{region '#Template'}
	{attribute 'Version' := '1.0.0.0'}
	{attribute 'Tags' := '"LCID": "1031", "Text": "Universal, Control, Scaling"'}
	{attribute 'Tags' := '"LCID": "1033", "Text": "Universal, Control, Scaling"'}
	{attribute 'Description' := '"LCID": "1031", "Text": "Skalierung"'}
	{attribute 'Description' := '"LCID": "1033", "Text": "Scaling"'}
{endregion}
FUNCTION_BLOCK FB_BA_Scale_02 EXTENDS FB_BA_View
VAR_INPUT
	fX			: REAL;
END_VAR
VAR_OUTPUT
	fY			: REAL;
END_VAR
VAR_INPUT CONSTANT
	X1			: FB_BA_AV_Op;	
	X2			: FB_BA_AV_Op;	
	Y1			: FB_BA_AV_Op;	
	Y2			: FB_BA_AV_Op;	
	YMin		: FB_BA_AV_Op;			
	YMax		: FB_BA_AV_Op;											   
	Y			: FB_BA_AV_Op;		
END_VAR
VAR
	Scale		: FB_BA_Chrct02;
END_VAR

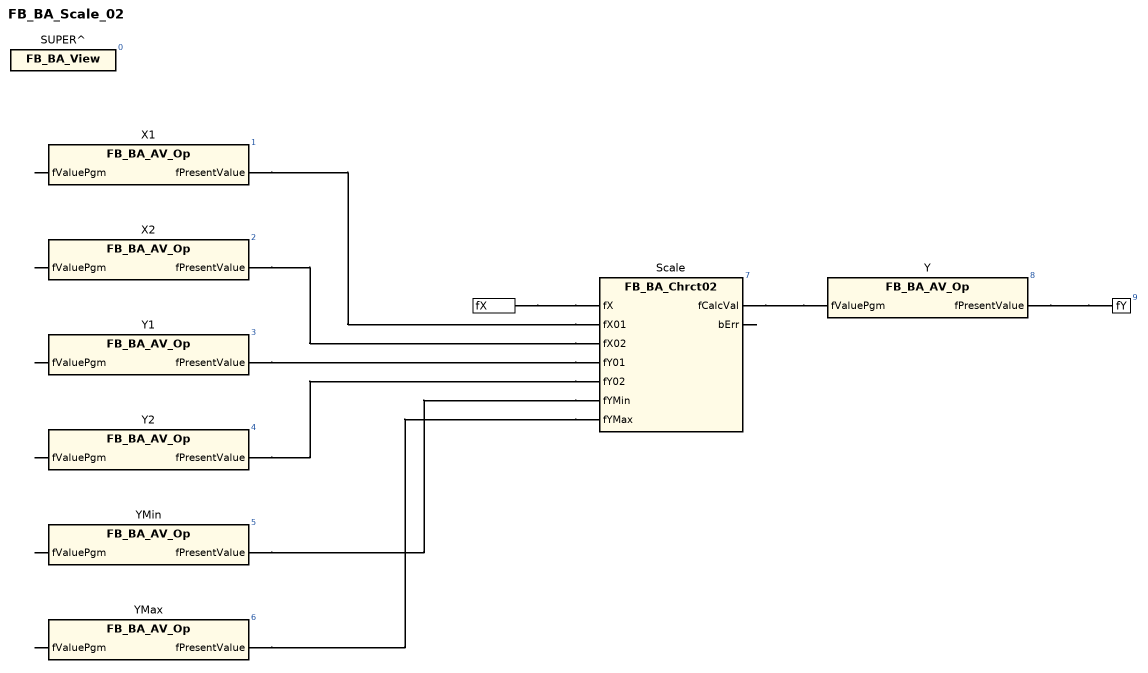
SUPER^(); // FB_BA_View
X1(); // FB_BA_AV_Op
X2(); // FB_BA_AV_Op
Y1(); // FB_BA_AV_Op
Y2(); // FB_BA_AV_Op
YMin(); // FB_BA_AV_Op
YMax(); // FB_BA_AV_Op
Scale(
    fX := fX,
    fX01 := X1.fPresentValue,
    fX02 := X2.fPresentValue,
    fY01 := Y1.fPresentValue,
    fY02 := Y2.fPresentValue,
    fYMin := YMin.fPresentValue,
    fYMax := YMax.fPresentValue); // FB_BA_Chrct02
Y(fValuePgm := Scale.fCalcVal); // FB_BA_AV_Op
fY := Y.fPresentValue;

METHOD FB_init : BOOL
VAR_INPUT
	bInitRetains : BOOL; // if TRUE, the retain variables are initialized (warm start / cold start)
	bInCopyCode : BOOL;  // if TRUE, the instance afterwards gets moved into the copy code (online change)
END_VAR
X1.iParent			:= THIS^;
X1.iLabel			:= LblUniControl.Scale_X01;	
X1.sObjectName		:= '{Idx=01}';		
X1.eUnit			:= E_BA_Unit.eTemperature_DegreesCelsius;						 	 
X1.fValueRm			:= -10.0;
X1.fCOVIncrement	:= BA2_Param.fDefCOVIncrement;		

X2.iParent			:= THIS^;
X2.iLabel			:= LblUniControl.Scale_X02;							
X2.sObjectName		:= '{Idx=02}';								 	 
X2.eUnit			:= E_BA_Unit.eTemperature_DegreesCelsius;						 	 
X2.fValueRm			:= -20.0;
X2.fCOVIncrement	:= BA2_Param.fDefCOVIncrement;		

Y1.iParent			:= THIS^;
Y1.iLabel			:= LblUniControl.Scale_Y01;							
Y1.sObjectName		:= '{Idx=01}';								 	 
Y1.eUnit			:= E_BA_Unit.eTemperature_DegreesCelsius;						 	 
Y1.fValueRm			:= 25.0;
Y1.fCOVIncrement	:= BA2_Param.fDefCOVIncrement;		
	
Y2.iParent			:= THIS^;
Y2.iLabel			:= LblUniControl.Scale_Y02;	
Y2.sObjectName		:= '{Idx=02}';								 	 
Y2.eUnit			:= E_BA_Unit.eTemperature_DegreesCelsius;						 	 
Y2.fValueRm			:= 40.0;
Y2.fCOVIncrement	:= BA2_Param.fDefCOVIncrement;		

YMin.iParent		:= THIS^;
YMin.iLabel			:= LblUniControl.Scale_Ymin;		
YMin.sObjectName	:= '{Idx=01}';								 	 
YMin.eUnit			:= E_BA_Unit.eTemperature_DegreesCelsius;						 	 
YMin.fValueRm		:= 10.0;
YMin.fCOVIncrement	:= BA2_Param.fDefCOVIncrement;		

YMax.iParent		:= THIS^;
YMax.iLabel			:= LblUniControl.Scale_Ymax;	
YMax.sObjectName	:= '{Idx=01}';								 	 
YMax.eUnit			:= E_BA_Unit.eTemperature_DegreesCelsius;						 	 
YMax.fValueRm		:= 60.0;
YMax.fCOVIncrement	:= BA2_Param.fDefCOVIncrement;		

Y.iParent			:= THIS^;
Y.iLabel			:= LblUniControl.Scale_Y;					
Y.sObjectName		:= '{Idx=01}';								 	 
Y.eUnit				:= E_BA_Unit.eTemperature_DegreesCelsius;						 	 		
Y.fCOVIncrement		:= BA2_Param.fDefCOVIncrement;
END_METHOD

METHOD GetPoint : BOOL
VAR_INPUT
	nIndex		: INT;
END_VAR
VAR_OUTPUT
	fbObjectX	: I_BA_AnalogOpObject;
	fbObjectY	: I_BA_AnalogOpObject;
END_VAR
CASE (nIndex) OF
	1:
		fbObjectX := X1;
		fbObjectY := Y1;
	2:
		fbObjectX := X2;
		fbObjectY := Y2;
ELSE
	RETURN;
END_CASE

GetPoint := TRUE;
END_METHOD

END_FUNCTION_BLOCK

(* stored: Version 1.1.0.1, ProductVersion 3.1.4024.9
   POU FB_BA_Scale_02: Id {0ff5bbf8-98e7-4a74-8fd1-b814991b4289}, SpecialFunc None
   Folder Management: Id {b33db001-b086-49c1-9c61-dede7ffea175}
   Method FB_init: Id {2c94549f-0d49-47a5-a361-c29623326ea0}
   Method GetPoint: Id {ea4c0245-eebb-4eeb-a7f6-83ff1ae6b9a3} *)
